FUNCTION_BLOCK FB_ConveyorLogSequence IMPLEMENTS I_ConveyorSequence
VAR_INPUT
END_VAR
VAR_OUTPUT
END_VAR
VAR
	nStep : UINT;
END_VAR


METHOD M_ConveyorSequence : BOOL
VAR_INPUT
	in_rConveyor	: REFERENCE TO FB_Conveyor;
END_VAR
CASE nStep OF
	0: 
		IF in_rConveyor.in_bStart THEN
			in_rConveyor.in_bStart := FALSE;
			in_rConveyor.M_StartConveyor();
			nStep := 10;
		END_IF
		
	10: 
		IF in_rConveyor.out_fbSensorSignal.GetTriggerSignal THEN
			fbLogList.M_Warning(
				in_iModule:=in_rConveyor,
				in_sMessage:='Material erfasst!'	
			);
		END_IF
		
		IF in_rConveyor.in_bStop THEN
			in_rConveyor.in_bStop := FALSE;
			in_rConveyor.M_StopConveyor();
			nStep := 20;
		END_IF
 
	20:
		
		nStep := 30;
	
	30:
	
END_CASE
END_METHOD

END_FUNCTION_BLOCK

(* stored: Version 1.1.0.1, ProductVersion 3.1.4022.16
   POU FB_ConveyorLogSequence: Id {c7d7066e-2f5b-4868-9d6e-b1f392a4abcb}, SpecialFunc None
   Method M_ConveyorSequence: Id {a7299fa3-e080-4d5f-b90b-062f9b103495} *)
